# EPICS substitutions: db/user.substitutions
# Example substitutions file

file "db/dbExample1.db" {
    { user = "crispd" }
}

file db/dbExample2.db {
    pattern { user, no, scan }
        { "crispd", 1, "1 second" }
        { "crispd", 2, "2 second" }
        { "crispd", 3, "5 second" }
}
